TYPE AxesRotationAxisParts :
STRUCT
	///The virtual axis
	virtualAxis: AngularAxis;
	///The physical axis
	physicalAxis: AngularAxis;
END_STRUCT
END_TYPE

(* stored: Version 1.1.0.1, ProductVersion 3.1.4019.2
   DUT AxesRotationAxisParts: Id {173f0ac0-3a86-4e48-b050-68a4a7055254} *)
